// Mitsubishi GX Works2 project: Rev - 18-03-19   PLC: Q00J

PROGRAM MAIN
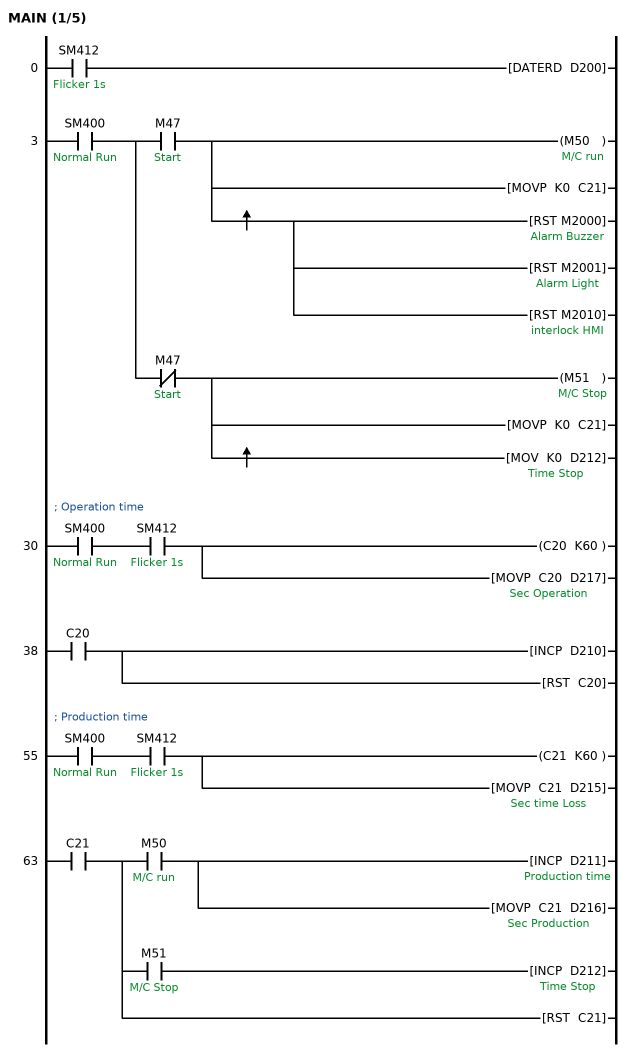
0     LD      SM412  ; Flicker 1s
      DATERD  D200
3     LD      SM400  ; Normal Run
      MPS
      AND     M47  ; Start
      OUT     M50  ; M/C run
      MOVP    K0 C21
      MEP
      RST     M2000  ; Alarm Buzzer
      RST     M2001  ; Alarm Light
      RST     M2010  ; interlock HMI
      MPP
      ANI     M47  ; Start
      OUT     M51  ; M/C Stop
      MOVP    K0 C21
      MEP
      MOV     K0 D212  ; Time Stop
; Operation time
30    LD      SM400  ; Normal Run
      AND     SM412  ; Flicker 1s
      OUT     C20 K60
      MOVP    C20 D217  ; Sec Operation
38    LD      C20
      INCP    D210
      RST     C20
; Production time
55    LD      SM400  ; Normal Run
      AND     SM412  ; Flicker 1s
      OUT     C21 K60
      MOVP    C21 D215  ; Sec time Loss
63    LD      C21
      MPS
      AND     M50  ; M/C run
      INCP    D211  ; Production time
      MOVP    C21 D216  ; Sec Production
      MRD
      AND     M51  ; M/C Stop
      INCP    D212
      MPP
      RST     C21
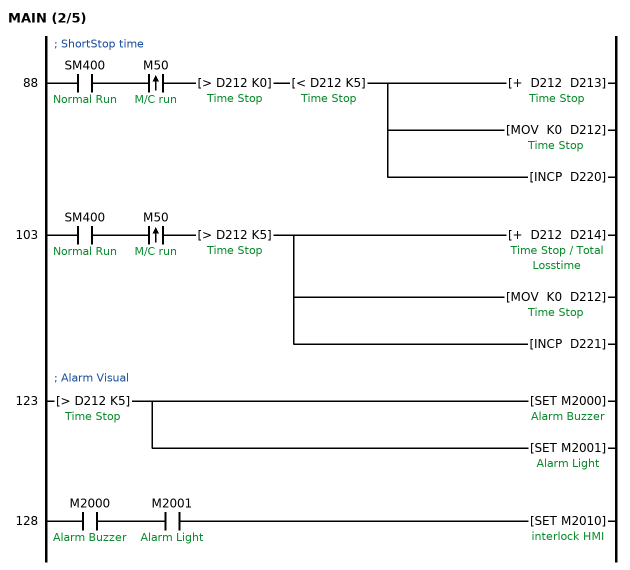
; ShortStop time
88    LD      SM400  ; Normal Run
      ANDP    M50  ; M/C run
      AND>    D212 K0  ; Time Stop
      AND<    D212 K5  ; Time Stop
      +       D212 D213
      MOV     K0 D212
      INCP    D220
103   LD      SM400  ; Normal Run
      ANDP    M50  ; M/C run
      AND>    D212 K5  ; Time Stop
      +       D212 D214  ; Total Losstime
      MOV     K0 D212
      INCP    D221
; Alarm Visual
123   LD>     D212 K5  ; Time Stop
      SET     M2000  ; Alarm Buzzer
      SET     M2001  ; Alarm Light
128   LD      M2000  ; Alarm Buzzer
      AND     M2001  ; Alarm Light
      SET     M2010  ; interlock HMI
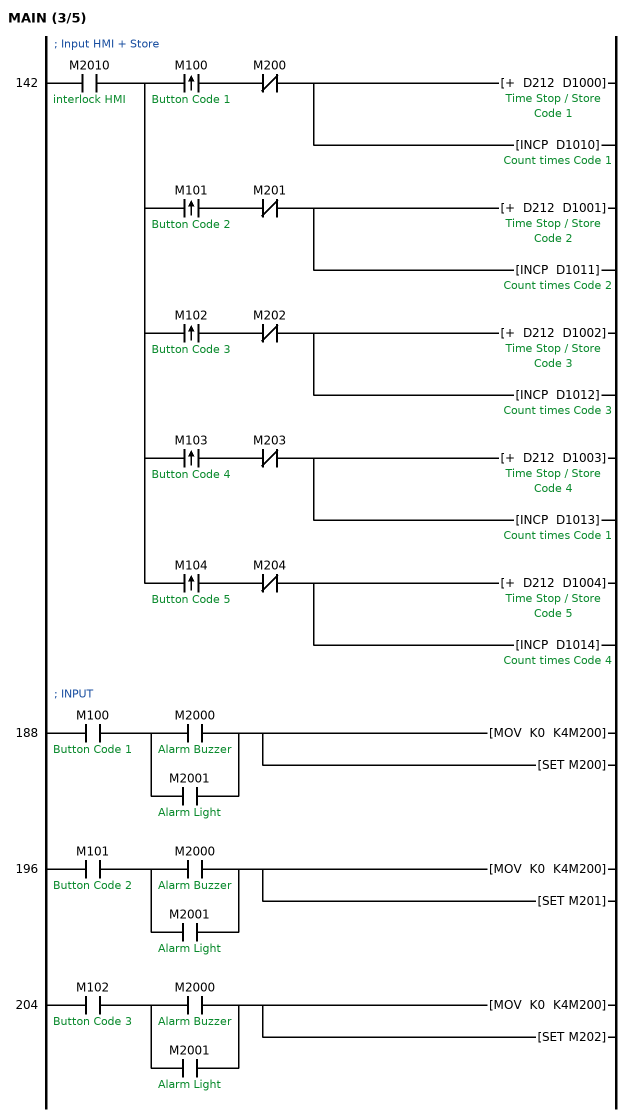
; Input HMI + Store
142   LD      M2010  ; interlock HMI
      MPS
      ANDP    M100  ; Button Code 1
      ANI     M200
      +       D212 D1000  ; Store Code 1
      INCP    D1010  ; Count times Code 1
      MRD
      ANDP    M101  ; Button Code 2
      ANI     M201
      +       D212 D1001  ; Store Code 2
      INCP    D1011  ; Count times Code 2
      MRD
      ANDP    M102  ; Button Code 3
      ANI     M202
      +       D212 D1002  ; Store Code 3
      INCP    D1012  ; Count times Code 3
      MRD
      ANDP    M103  ; Button Code 4
      ANI     M203
      +       D212 D1003  ; Store Code 4
      INCP    D1013  ; Count times Code 1
      MPP
      ANDP    M104  ; Button Code 5
      ANI     M204
      +       D212 D1004  ; Store Code 5
      INCP    D1014  ; Count times Code 4
; INPUT
188   LD      M100  ; Button Code 1
      LD      M2000  ; Alarm Buzzer
      OR      M2001  ; Alarm Light
      ANB
      MOV     K0 K4M200
      SET     M200
196   LD      M101  ; Button Code 2
      LD      M2000  ; Alarm Buzzer
      OR      M2001  ; Alarm Light
      ANB
      MOV     K0 K4M200
      SET     M201
204   LD      M102  ; Button Code 3
      LD      M2000  ; Alarm Buzzer
      OR      M2001  ; Alarm Light
      ANB
      MOV     K0 K4M200
      SET     M202
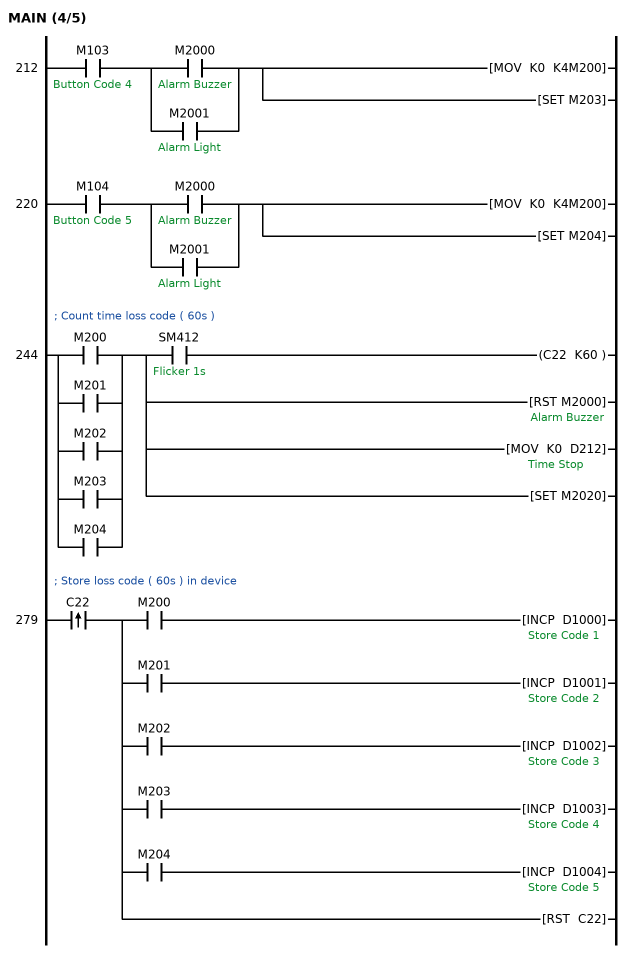
212   LD      M103  ; Button Code 4
      LD      M2000  ; Alarm Buzzer
      OR      M2001  ; Alarm Light
      ANB
      MOV     K0 K4M200
      SET     M203
220   LD      M104  ; Button Code 5
      LD      M2000  ; Alarm Buzzer
      OR      M2001  ; Alarm Light
      ANB
      MOV     K0 K4M200
      SET     M204
; Count time loss code ( 60s )
244   LD      M200
      OR      M201
      OR      M202
      OR      M203
      OR      M204
      MPS
      AND     SM412  ; Flicker 1s
      OUT     C22 K60
      MPP
      RST     M2000  ; Alarm Buzzer
      MOV     K0 D212
      SET     M2020
; Store loss code ( 60s ) in device
279   LDP     C22
      MPS
      AND     M200
      INCP    D1000
      MRD
      AND     M201
      INCP    D1001
      MRD
      AND     M202
      INCP    D1002
      MRD
      AND     M203
      INCP    D1003
      MRD
      AND     M204
      INCP    D1004
      MPP
      RST     C22
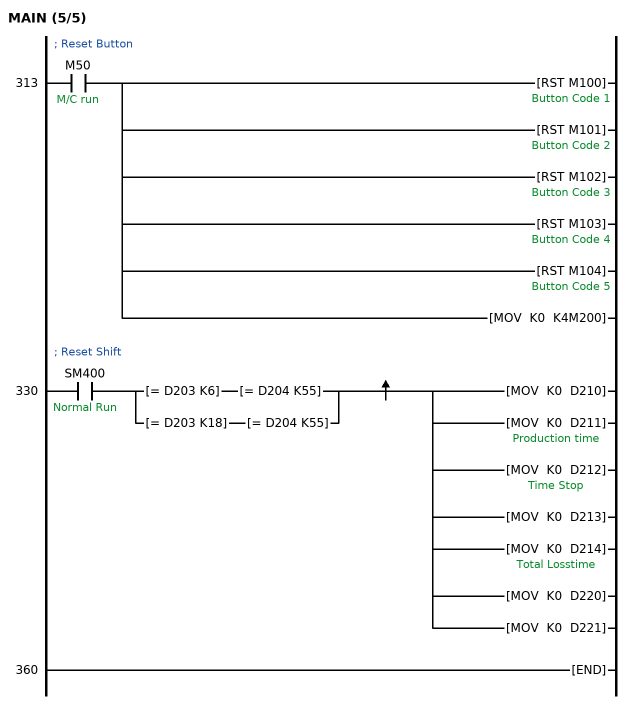
; Reset Button
313   LD      M50  ; M/C run
      RST     M100  ; Button Code 1
      RST     M101  ; Button Code 2
      RST     M102  ; Button Code 3
      RST     M103  ; Button Code 4
      RST     M104  ; Button Code 5
      MOV     K0 K4M200
; Reset Shift
330   LD      SM400  ; Normal Run
      LD=     D203 K6
      AND=    D204 K55
      LD=     D203 K18
      AND=    D204 K55
      ORB
      ANB
      MEP
      MOV     K0 D210
      MOV     K0 D211
      MOV     K0 D212
      MOV     K0 D213
      MOV     K0 D214
      MOV     K0 D220
      MOV     K0 D221
360   END
END_PROGRAM
